{attribute 'qualified_only'}
VAR_GLOBAL
	counter : DINT;
	origin : ST_Point;
	mode : E_Mode := E_Mode.Idle;
END_VAR

(* stored: Version 1.1.0.1, ProductVersion 3.1.4026.18
   GVL GVL_Main: Id {00000000-0000-0000-0000-000000000010} *)
